FUNCTION_BLOCK FB_CsvPersistentEventStorage IMPLEMENTS I_PersistentEventStorage
VAR_INPUT
	fbFileOpen : FB_FileOpen := (sPathName := 'C:\Events.log', nMode := FOPEN_MODEAPPEND OR FOPEN_MODETEXT);
	fbFilePuts : FB_FilePuts;
	fbFileClose : FB_FileClose;
	eWriteState : (FILE_OPEN_TRIGGER, FILE_OPEN, WAIT_FOR_EVENT, WRITE_EVENT_TRIGGER, WRITE_EVENT, FILE_CLOSE_TRIGGER, FILE_CLOSE, ERROR);
	stEventWrittenToFile : ST_Event;
	CsvString : T_MaxString;
	FILE_CLOSE_TRIGGER : INT;
END_VAR
VAR_OUTPUT
END_VAR
VAR
	FILE_CLOSE: INT;
END_VAR

CASE eWriteState OF
	FILE_OPEN_TRIGGER:
		fbFileOpen(bExecute := TRUE);
		eWriteState := FILE_OPEN;
	
	FILE_OPEN:
		fbFileOpen(bExecute := FALSE);
		IF fbFileOpen.bError THEN
			eWriteSTate := ERROR;
		ELSIF NOT fbFileOpen.bBusy AND fbFileOpen.hFile <> 0 THEN
			eWriteState := WAIT_FOR_eVENT;
		END_IF
		
	WAIT_FOR_EVENT:
		//do nothing
		
	WRITE_EVENT_TRIGGER:
		CsvString := CreateCsvString(stEvent := stEventWrittenToFile);
		fbFilePuts(bExecute := TRUE,
					sLine := CsvString,
					hFile := fbFileOpen.hFile);
			
	FILE_CLOSE_TRIGGER:
		fbFileClose(bExecute := TRUE,
					hFile := fbFileOpen.hFile);
		eWriteState := FILE_CLOSE;
		
	FILE_CLOSE:
		fbFileClose(bExecute := FALSE);
		IF fbFileClose.bError THEN
			eWriteState := ERROR;
		ELSIF NOT fbFileClose.bBusy THEN
			eWriteState := FILE_OPEN_TRIGGER;
		END_IF
		
	ERROR:
		//DO NOTHING
END_CASE

METHOD CreateCsvString : T_MaxString
VAR_INPUT
	stEvent : REFERENCE TO ST_Event;
END_VAR
VAR
	TempString : T_MaxString;
END_VAR
TempString := TO_STRING(stEvent.eEventType);
TempString := CONCAT(STR1 := TempString, STR2 := ',');
TempString := CONCAT(STR1 := TempString, STR2 := TO_STRING(stEvent.eEventSeverity));
TempString := CONCAT(STR1 := TempString, STR2 := ',');
TempString := CONCAT(STR1 := TempString, STR2 := TO_STRING(stEvent.nEventIdentity));
TempString := CONCAT(STR1 := TempString, STR2 := ',');
TempString := CONCAT(STR1 := TempString, STR2 := stEvent.sEventText);
TempString := CONCAT(STR1 := TempString, STR2 := ',');
TempString := CONCAT(STR1 := TempString, STR2 := TO_STRING(stEvent.dtTimestamp));
TempString := CONCAT(STR1 := TempString, STR2 := '$n');

CreateCsvString := TempString;
END_METHOD

METHOD StoreEvent
VAR_INPUT
	stEvent	: ST_Event;
END_VAR
IF eWriteState = WAIT_FOR_EVENT THEN
	eWriteState := WRITE_EVENT_TRIGGER;
	stEventWrittenToFile := stEvent;
END_IF
END_METHOD

END_FUNCTION_BLOCK

(* stored: Version 1.1.0.1, ProductVersion 3.1.4024.12
   POU FB_CsvPersistentEventStorage: Id {ce4c8058-680e-4e4f-9bfe-931fd5000886}, SpecialFunc None
   Method CreateCsvString: Id {95beddc0-7941-4c10-8070-7f190cb5b048}
   Method StoreEvent: Id {1ac76475-49cf-4a66-85dd-3eeceb2634d0} *)
